PROGRAM JoystickTimeout
VAR
	 preReceiveCount:UINT;
END_VAR

IF preReceiveCount<>receive_counter3 THEN
	joyStickInfoIns.CommunictionStatus:=1;
ELSE
	joyStickInfoIns.CommunictionStatus:=0;
END_IF
preReceiveCount:=receive_counter3;

END_PROGRAM

(* stored: Version 1.1.0.1, ProductVersion 3.1.4018.2
   POU JoystickTimeout: Id {f5a01ca4-271a-404d-b50d-23c26e5b38b0}, SpecialFunc None *)
